ABB RobotStudio station: Gripper.rspag

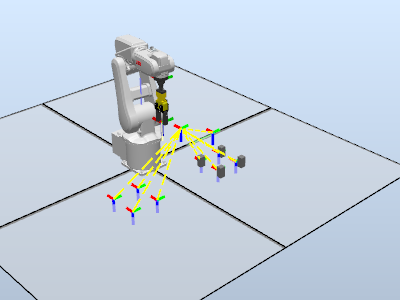
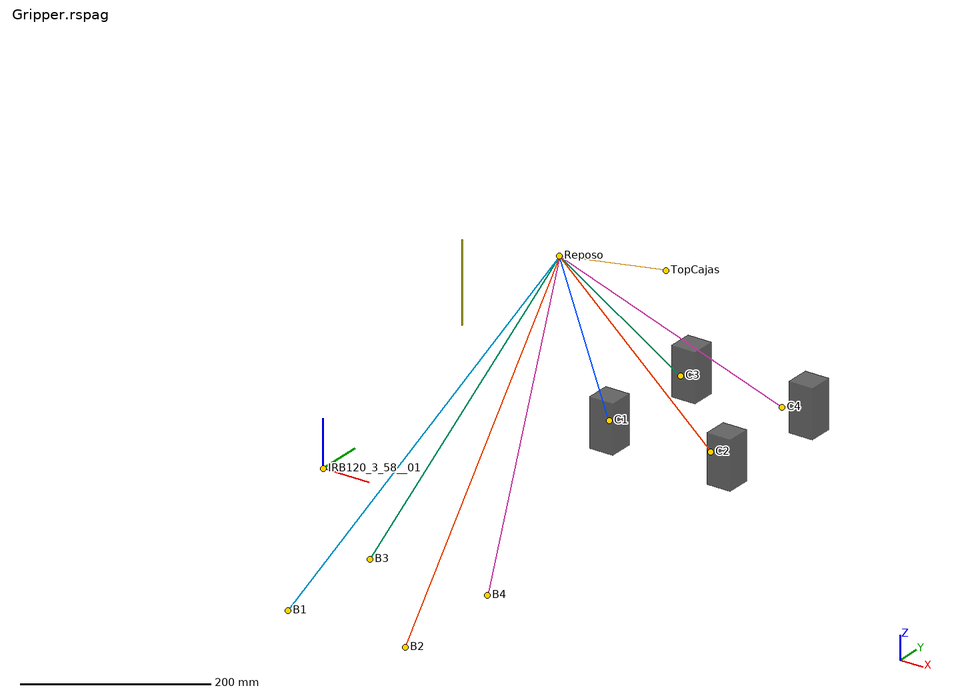
[picture v1: parts stored in the station drawn from their meshes, with robot base, taught points and paths (robot models come from the ABB library and are not in the file)]
--- station ---
Station Solution_IRB120 (saved by RobotStudio 22.2.9947.0)
Controller 120-500061
  mechanical unit ROB_1: IRB120_3_58__01, 6 joints, base frame (0, 0, 0) mm
Layout (positions relative to the parent item):
  - IRB120_3_58__01 [mechanism, from Robots\IRB120_3_58_G_01.rslib] at (0, 0, 0) mm; joint values [-0.7854, 0.254, 0.7782, 0, 0.5386, -0.7854] (rad or m)
  - caja2 [part], size 30 x 30 x 60 mm
  - caja3 [part], size 30 x 30 x 60 mm
  - caja4 [part], size 30 x 30 x 60 mm
  - caja1 [part], size 30 x 30 x 60 mm
  - SmartComponent_1 [smart component]
      signals: DI CogerCaja, DI SoltarCaja, DO SensorCaja
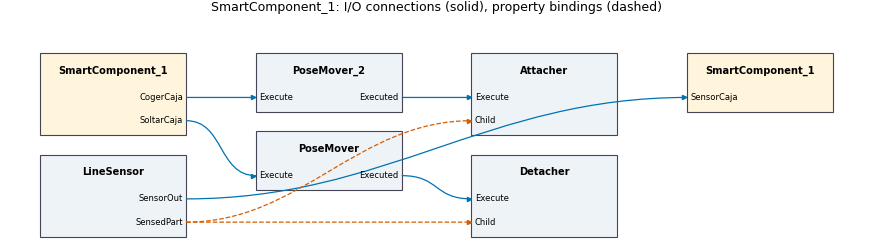
      connections:
        SmartComponent_1.CogerCaja -> PoseMover_2.Execute
        SmartComponent_1.SoltarCaja -> PoseMover.Execute
        PoseMover_2.Executed -> Attacher.Execute
        PoseMover.Executed -> Detacher.Execute
        LineSensor.SensorOut -> SmartComponent_1.SensorCaja
        LineSensor.SensedPart => Detacher.Child
        LineSensor.SensedPart => Attacher.Child
    - PoseMover [smart component, from Components\PoseMover.rslib]
        properties: Mechanism=gripper_SCHUNK_GWB44; Pose=2; Duration=0.5
    - gripper_SCHUNK_GWB44 [mechanism, from Herramientas\gripper_SCHUNK_GWB44.rslib] at (200, -32.01, 561.62) mm, rotated rx -180 ry 0 rz -180 deg; joint values [0, 0] (rad or m)
    - PoseMover_2 [smart component, from Components\PoseMover.rslib]
        properties: Mechanism=gripper_SCHUNK_GWB44; Pose=3; Duration=0.5
    - LineSensor [smart component, from Components\LineSensor.rslib] at (200, -32.01, 335.62) mm, rotated rx -180 ry 0 rz -180 deg
        properties: Start=[0 0 0]; End=[0 0 0.1]; Radius=0.0005; SensedPart=(none); SensedPoint=[0 0 0]
      - _sensorPart_ [part], size 1 x 1 x 100 mm
    - Attacher [smart component, from Components\Attacher.rslib] at (-430, -32.01, 935.62) mm, rotated rx -44.22 ry 90 rz -44.22 deg
        properties: Parent=gripper_SCHUNK_GWB44; Flange=0; Child=(none); Mount=false; Offset=[0 0 0]; Orientation=[0 0 0]
    - Detacher [smart component, from Components\Detacher.rslib]
        properties: Child=(none); KeepPosition=true
Attachment: gripper_SCHUNK_GWB44 is attached to IRB120_3_58__01 / Link6
Attachment: Attacher is attached to IRB120_3_58__01 / Link6
Attachment: LineSensor is attached to gripper_SCHUNK_GWB44 / L1
Station logic (signal -> signal, property => property):
  120-500061.CogerBote -> SmartComponent_1.CogerCaja
  120-500061.SoltarBote -> SmartComponent_1.SoltarCaja

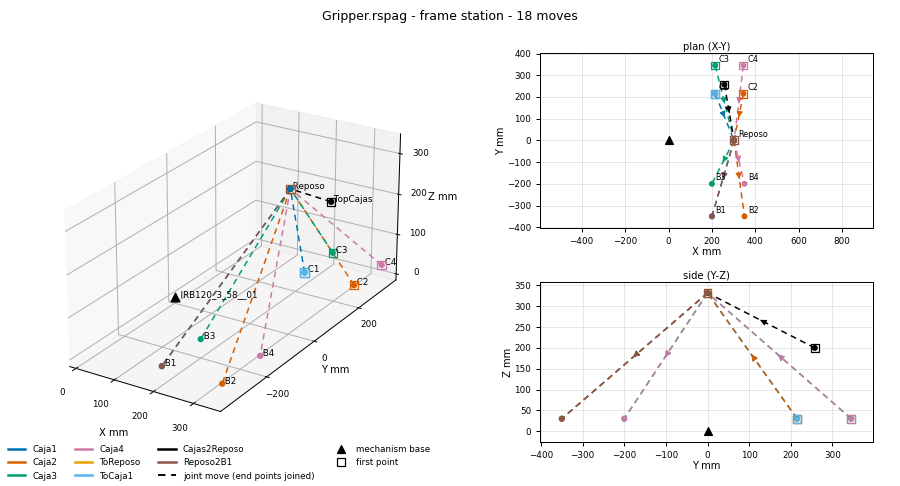
[picture p0: tool path of Gripper.rspag in frame station, 18 of 18 moves have a stored position in this frame; points joined in program order, loops and branches not executed]
--- Backups/120-500061/RAPID/TASK1/PROGMOD/CalibData.mod ---
MODULE CalibData
    PERS tooldata gripper_SCHUNK_GWB44:=[TRUE,[[0,0,226],[1,0,0,0]],[0.5,[0,0,110],[1,0,0,0],0,0,0]];
ENDMODULE

--- Backups/120-500061/RAPID/TASK1/PROGMOD/MainModule.mod ---
MODULE MainModule
	PROC main()
        SetDO DO10_11,1; !Abrir el gripper
        SetDO DO10_10,0;!No cerrar el gripper
        ToReposo;

        !Caja1
        Caja1;
        WaitTime 1;
        SetDO DO10_11,0;
        SetDO DO10_10,1; !Cierra gripper
        SetDO CogerBote,1;
        SetDO CogerBote,0;
        WaitTime 1;

        Cajas2Reposo;
        Reposo2B1;
        WaitTime 1;
        SetDO DO10_11,1;
        SetDO DO10_10,0;
        SetDO SoltarBote,1;
        SetDO SoltarBote,0;

        ToReposo;




	ENDPROC
ENDMODULE

--- Backups/120-500061/RAPID/TASK1/PROGMOD/Module1.mod ---
MODULE Module1

    CONST robtarget C1:=[[215,215,30],[0,0,1,0],[0,0,0,0],[9E+09,9E+09,9E+09,9E+09,9E+09,9E+09]];
    CONST robtarget Reposo:=[[302,0,332],[0,0,1,0],[0,0,0,0],[9E+09,9E+09,9E+09,9E+09,9E+09,9E+09]];
    CONST robtarget B1:=[[200,-350,30],[0,0,1,0],[0,0,0,0],[9E+09,9E+09,9E+09,9E+09,9E+09,9E+09]];
    CONST robtarget C2:=[[345,215,30],[0,0,1,0],[0,0,0,0],[9E+09,9E+09,9E+09,9E+09,9E+09,9E+09]];
    CONST robtarget B2:=[[350,-350,30],[0,0,1,0],[-1,0,-1,0],[9E+09,9E+09,9E+09,9E+09,9E+09,9E+09]];
    CONST robtarget C3:=[[215,345,30],[0,0,1,0],[0,0,0,0],[9E+09,9E+09,9E+09,9E+09,9E+09,9E+09]];
    CONST robtarget B3:=[[200,-200,30],[0,0,1,0],[0,0,0,0],[9E+09,9E+09,9E+09,9E+09,9E+09,9E+09]];
    CONST robtarget C4:=[[345,345,30],[0,0,1,0],[0,0,0,0],[9E+09,9E+09,9E+09,9E+09,9E+09,9E+09]];
    CONST robtarget B4:=[[350,-200,30],[0,0,1,0],[-1,0,-1,0],[9E+09,9E+09,9E+09,9E+09,9E+09,9E+09]];
    CONST robtarget TopCajas:=[[257.5,257.5,200],[0,0,1,0],[0,0,0,0],[9E+09,9E+09,9E+09,9E+09,9E+09,9E+09]];

    PROC Caja1()
        MoveJ C1,v200,fine,gripper_SCHUNK_GWB44\WObj:=wobj0;
        MoveJ Reposo,v200,fine,gripper_SCHUNK_GWB44\WObj:=wobj0;
        MoveJ B1,v200,fine,gripper_SCHUNK_GWB44\WObj:=wobj0;
    ENDPROC
    PROC Caja2()
        MoveJ C2,v200,fine,gripper_SCHUNK_GWB44\WObj:=wobj0;
        MoveJ Reposo,v200,fine,gripper_SCHUNK_GWB44\WObj:=wobj0;
        MoveJ B2,v200,fine,gripper_SCHUNK_GWB44\WObj:=wobj0;
    ENDPROC
    PROC Caja3()
        MoveJ C3,v200,fine,gripper_SCHUNK_GWB44\WObj:=wobj0;
        MoveJ Reposo,v200,fine,gripper_SCHUNK_GWB44\WObj:=wobj0;
        MoveJ B3,v200,fine,gripper_SCHUNK_GWB44\WObj:=wobj0;
    ENDPROC
    PROC Caja4()
        MoveJ C4,v200,fine,gripper_SCHUNK_GWB44\WObj:=wobj0;
        MoveJ Reposo,v200,fine,gripper_SCHUNK_GWB44\WObj:=wobj0;
        MoveJ B4,v200,fine,gripper_SCHUNK_GWB44\WObj:=wobj0;
    ENDPROC
    PROC ToReposo()
        MoveJ Reposo,v200,fine,gripper_SCHUNK_GWB44\WObj:=wobj0;
    ENDPROC
    PROC ToCaja1()
        MoveJ C1,v200,fine,gripper_SCHUNK_GWB44\WObj:=wobj0;
    ENDPROC
    PROC Cajas2Reposo()
        MoveJ TopCajas,v200,fine,gripper_SCHUNK_GWB44\WObj:=wobj0;
        MoveJ Reposo,v200,fine,gripper_SCHUNK_GWB44\WObj:=wobj0;
    ENDPROC
    PROC Reposo2B1()
        MoveJ Reposo,v200,fine,gripper_SCHUNK_GWB44\WObj:=wobj0;
        MoveJ B1,v200,fine,gripper_SCHUNK_GWB44\WObj:=wobj0;
    ENDPROC
ENDMODULE

--- Backups/120-500061/SYSPAR/EIO.cfg ---
EIO:CFG_1.0:5:0::
#
EIO_BUS:

      -Name "Virtual1" -ConnectorID "SIM1"

      -Name "DeviceNet_Lean" -BusType "DNLE" -ConnectorID "PCI1"\
      -ConnectorLabel "DeviceNet Lean"
#
EIO_UNIT_TYPE:

      -Name "Virtual" -VendorName "ABB" -ProductName "Virtual unit"

      -Name "d651_Lean" -BusType "DNLE" -VendorName "ABB Robotics"\
      -ProductName "Combi Unit" -DL_ProductCode 25

      -Name "d652_Lean" -BusType "DNLE" -VendorName "ABB Robotics"\
      -ProductName "24 VDC Unit" -DL_ProductCode 26

      -Name "d653_Lean" -BusType "DNLE" -VendorName "ABB Robotics"\
      -ProductName "Relay Unit" -DL_ProductCode 27

      -Name "AC500_PLC_Lean" -BusType "DNLE" -VendorName "ABB Stotz"\
      -ProductName "AC500 PLC - FPB" -DL_ProductCode 1 -DL_VendorID 760

      -Name "DL_GENERIC" -BusType "DNLE" -DL_ProductCode 3535

      -Name "DL_GENERIC_POLL" -BusType "DNLE" -DL_ProductCode 3535\
      -DL_Pollrate 30

      -Name "d351_Lean" -BusType "DNLE" -VendorName "ABB Robotics"\
      -ProductName "IBS Adapter" -DL_ProductCode 7

      -Name "d378_Lean" -BusType "DNLE" -VendorName "ABB Robotics"\
      -ProductName "CCLink Adapter" -DL_ProductCode 17
#
EIO_UNIT:

      -Name "BOARD10" -UnitType "d652_Lean" -Bus "DeviceNet_Lean" -DL_Address 10

      -Name "ABB" -UnitType "Virtual" -Bus "Virtual1"
#
EIO_SIGNAL:

      -Name "DI10_1" -SignalType "DI" -Unit "BOARD10" -UnitMap "0"

      -Name "DI10_2" -SignalType "DI" -Unit "BOARD10" -UnitMap "1"

      -Name "DI10_3" -SignalType "DI" -Unit "BOARD10" -UnitMap "2"

      -Name "DI10_4" -SignalType "DI" -Unit "BOARD10" -UnitMap "3"

      -Name "DI10_5" -SignalType "DI" -Unit "BOARD10" -UnitMap "4"

      -Name "DI10_6" -SignalType "DI" -Unit "BOARD10" -UnitMap "5"

      -Name "DI10_7" -SignalType "DI" -Unit "BOARD10" -UnitMap "6"

      -Name "DI10_8" -SignalType "DI" -Unit "BOARD10" -UnitMap "7"

      -Name "DI10_9" -SignalType "DI" -Unit "BOARD10" -UnitMap "8"

      -Name "DI10_10" -SignalType "DI" -Unit "BOARD10" -UnitMap "9"

      -Name "DI10_11" -SignalType "DI" -Unit "BOARD10" -UnitMap "10"

      -Name "DI10_12" -SignalType "DI" -Unit "BOARD10" -UnitMap "11"

      -Name "DI10_13" -SignalType "DI" -Unit "BOARD10" -UnitMap "12"

      -Name "DI10_14" -SignalType "DI" -Unit "BOARD10" -UnitMap "13"

      -Name "DI10_15" -SignalType "DI" -Unit "BOARD10" -UnitMap "14"

      -Name "DI10_16" -SignalType "DI" -Unit "BOARD10" -UnitMap "15"

      -Name "DO10_1" -SignalType "DO" -Unit "BOARD10" -UnitMap "0"

      -Name "DO10_2" -SignalType "DO" -Unit "BOARD10" -UnitMap "1"

      -Name "DO10_3" -SignalType "DO" -Unit "BOARD10" -UnitMap "2"

      -Name "DO10_4" -SignalType "DO" -Unit "BOARD10" -UnitMap "3"

      -Name "DO10_5" -SignalType "DO" -Unit "BOARD10" -UnitMap "4"

      -Name "DO10_6" -SignalType "DO" -Unit "BOARD10" -UnitMap "5"

      -Name "DO10_7" -SignalType "DO" -Unit "BOARD10" -UnitMap "6"

      -Name "DO10_8" -SignalType "DO" -Unit "BOARD10" -UnitMap "7"

      -Name "DO10_9" -SignalType "DO" -Unit "BOARD10" -UnitMap "8"

      -Name "DO10_10" -SignalType "DO" -Unit "BOARD10" -UnitMap "9"

      -Name "DO10_11" -SignalType "DO" -Unit "BOARD10" -UnitMap "10"

      -Name "DO10_12" -SignalType "DO" -Unit "BOARD10" -UnitMap "11"

      -Name "DO10_13" -SignalType "DO" -Unit "BOARD10" -UnitMap "12"

      -Name "DO10_14" -SignalType "DO" -Unit "BOARD10" -UnitMap "13"

      -Name "DO10_15" -SignalType "DO" -Unit "BOARD10" -UnitMap "14"

      -Name "DO10_16" -SignalType "DO" -Unit "BOARD10" -UnitMap "15"

      -Name "CogerBote" -SignalType "DO" -Unit "ABB" -UnitMap "1"

      -Name "SoltarBote" -SignalType "DO" -Unit "ABB" -UnitMap "2"
#
EIO_COMMAND_TYPE:

      -Name "StationNo_L" -UnitType "d378_Lean" -DefValue "1" -OrderNr 1\
      -DL_Path "6,20 68 24 01 30 01,C6,1" -DL_Service 16

      -Name "BaudRate_L" -UnitType "d378_Lean" -DefValue "0" -OrderNr 2\
      -DL_Path "6,20 68 24 01 30 02,C6,1" -DL_Service 16

      -Name "OccStat_L" -UnitType "d378_Lean" -DefValue "1" -OrderNr 3\
      -DL_Path "6,20 68 24 01 30 03,C6,1" -DL_Service 16

      -Name "BasicIO_L" -UnitType "d378_Lean" -DefValue "0" -OrderNr 4\
      -DL_Path "6,20 68 24 01 30 04,C1,1" -DL_Service 16

      -Name "D378reset_L" -UnitType "d378_Lean" -DefValue "0" -OrderNr 5\
      -DL_Path "4,20 01 24 01,C1,1" -DL_Service 5

      -Name "DataWidth_L" -UnitType "d351_Lean" -DefValue "3" -OrderNr 1\
      -DL_Path "6,20 65 24 01 30 01,C6,1" -DL_Service 16

      -Name "D351reset_L" -UnitType "d351_Lean" -DefValue "0" -OrderNr 2\
      -DL_Path "4,20 01 24 01,C1,1" -DL_Service 5
#
EIO_ACCESS:

      -Name "All" -Rapid  -LocalManual  -LocalAuto  -RemoteManual  -RemoteAuto

--- Backups/120-500061/SYSPAR/PROC.cfg ---
PROC:CFG_1.0:5:0::
#
GAP_TASK_NAME_MAPPING:

      -name "T_ROB1" -common_name "T_ROB1" -tab_index 1
